// TIA Portal V20 export
DATA_BLOCK "PM4"   // DB278
// stored: MemoryReserve 100
   VAR
      "TOP TAPE Clamp TOP LEFT UP" : Bool;
      "TOP TAPE Clamp TOP LEFT DOWN" : Bool;
      "TOP TAPE Clamp TOP CENTER UP" : Bool;
      "TOP TAPE Clamp TOP CENTER DOWN" : Bool;
      "TOP TAPE Clamp TOP RIGHT UP" : Bool;
      "TOP TAPE Clamp TOP RIGHT DOWN" : Bool;
      "TOP TAPE Clamp BTM UP" : Bool;
      "TOP TAPE Clamp BTM DOWN" : Bool;
      SPARE : Bool;
      SPARE_1 : Bool;
      SPARE_2 : Bool;
      SPARE_3 : Bool;
      SPARE_4 : Bool;
      SPARE_5 : Bool;
      SPARE_6 : Bool;
      SPARE_7 : Bool;
   END_VAR
BEGIN
END_DATA_BLOCK
